// TIA Portal V16 export
// export: Created 2024-09-05T17:39:24.7754954Z, ExportSetting WithDefaults, DisplayName Totally Integrated Automation Portal, DisplayVersion V16 Update 6, DisplayName TIA Portal Version Control Interface, DisplayVersion V16 Update 2, DisplayName TIA Portal Openness, DisplayVersion V16 Update 6, DisplayName STEP 7 Professional, DisplayVersion V16 Update 6, DisplayName STEP 7 Safety, DisplayVersion V16, DisplayName WinCC Advanced, DisplayVersion V16 Update 6
DATA_BLOCK "2. Call_M000_PRODUCTION_DECLARATION_DB"   // DB2003
AUTHOR : bartz
VERSION : 0.1
// stored: AutoNumber false, DBAccessibleFromOPCUA true, InstanceOfName 2. Call_M000_PRODUCTION_DECLARATION, InstanceOfType FB
"2. Call_M000_PRODUCTION_DECLARATION"
   // VAR_INPUT
   //    CYCLE_COUNTER : DInt;
   //    timeUTC { ExternalAccessible := 'False'; ExternalVisible := 'False'; ExternalWritable := 'False'} : DTL;
   // END_VAR
   // VAR_IN_OUT
   //    LOCAL_PART_ARRAY : Variant;
   //    LOCAL_PART_WSTRING : Variant;
   //    LOCAL_TOOL : Variant;
   //    TRACA_REF : Variant;
   //    QUANTITY : Variant;
   //    STATION_NAME : Variant;
   // END_VAR
   // VAR
   //    cycleCounter_temp : DInt;
   //    LOCAL_PART_OK : WString;
   //    STATION_NAME_OK : WString;
   //    datestring : WString;
   //    READ_TIMESTAMP : DTL;
   //    aux : Struct
   //       idx : UInt;
   //       cnt : UInt;
   //       sizeCnt : Bool;
   //       LOCAL_PART_STRING : String;
   //    END_STRUCT;
   // END_VAR
BEGIN
END_DATA_BLOCK
